(* CoDeSys 2.3 export: BR_ST.EXP *)

(* Data type *)
TYPE BR_ST :
	(
	BR_ERROR := 0,
	BR_SINS1_SELECTING,
	BR_SINS1_READY,
	BR_SINS2_SELECTING,
	BR_SINS2_READY,
	BR_YAG_SELECTING,
	BR_YAG_READY
	);
END_TYPE
